{attribute 'GeneratedUsingTerminal: EK1122-0000-0018'}
{attribute addProperty BoxType "EK1122-0000-0018"}
{attribute addProperty Id "Beckhoff_ELM3xxxsub_EK1100EK1100_AB5A94672"}
{attribute addProperty CRC "4096879235"}
{attribute addProperty Size "2"}
TYPE Beckhoff_ELM3xxxEK1122_F4316A83 EXTENDS EK1122_AB5A9467 :
STRUCT
	{attribute addProperty Name "Beckhoff_ELM3xxxsub_EK1100"}
	{attribute addProperty PreviousPort "Beckhoff ELM3xxxEK1122 : D"}
	Beckhoff_ELM3xxxsub_EK1100 : EK1100_AB5A9467;
END_STRUCT
END_TYPE

(* stored: Version 1.2.0.0, ProductVersion 3.1.4024.9
   DUT Beckhoff_ELM3xxxEK1122_F4316A83: Id {f430fc7c-f3e0-4b7b-99e6-ea02d2051b63} *)
